FUNCTION_BLOCK "Conversor_4-20_0-20"
{ S7_Optimized_Access := 'TRUE' }
VERSION : 0.1
   VAR_INPUT
      "IN_4-20" : Word;
   END_VAR

   VAR_OUTPUT
      "OUT_0-20" : Real;
   END_VAR


BEGIN
	#"OUT_0-20" := (#"IN_4-20" / 221.0) - 25.0;
END_FUNCTION_BLOCK

